FUNCTION_BLOCK InternalStorage EXTENDS TcoCore.TcoObject 
VAR
	_data : ARRAY [0..9] OF ProcessData := [(Parent := THIS^), (Parent := THIS^), (Parent := THIS^), (Parent := THIS^), (Parent := THIS^),
                                        (Parent := THIS^), (Parent := THIS^), (Parent := THIS^), (Parent := THIS^), (Parent := THIS^)];
END_VAR
VAR CONSTANT
	_maxNumberOfCarriers : UINT := 10;
END_VAR

METHOD GetByCarrier : BOOL
VAR_INPUT
	inCarrier : UINT;
END_VAR
VAR_IN_OUT
	inoData : ProcessData;
END_VAR
IF(inCarrier >= 0 AND inCarrier < _maxNumberOfCarriers) THEN
	inoData := _data[inCarrier];
	GetByCarrier := TRUE;
	RETURN;	
END_IF

Messenger.Post(CONCAT('<#Requested carrier is out of range of internal storage. Max number of carriers is#> ', UINT_TO_STRING(_maxNumberOfCarriers)), eMessageCategory.ProgrammingError);
END_METHOD

METHOD SaveByCarrier : BOOL
VAR_INPUT
	inCarrier : UINT;
END_VAR
VAR_IN_OUT
	inoData : ProcessData;
END_VAR
IF(inCarrier >= 0 AND inCarrier < _maxNumberOfCarriers) THEN
	_data[inCarrier] := inoData;
	SaveByCarrier := TRUE;
	RETURN;	
END_IF

Messenger.Post(CONCAT('<#Requested carrier is out of range of internal storage. Max number of carriers is#> ', UINT_TO_STRING(_maxNumberOfCarriers)), eMessageCategory.ProgrammingError);
END_METHOD

END_FUNCTION_BLOCK

(* stored: Version 1.1.0.1
   POU InternalStorage: Id {534e0d35-48f7-4157-8269-593be69f0ce5}, SpecialFunc None
   Method GetByCarrier: Id {301065f4-d903-4b59-8a60-be8ba9d252a8}
   Method SaveByCarrier: Id {3a2f772b-82f7-4e77-b628-277cfa0b1f34} *)
